Fanuc KAREL source: kb00143.KL

-- PROVISIONAL review KL for V1013-1; original PC SHA256 70a769824f0bb04e627808649afede2e4c1abad04249343c2b344672b59b27b0
-- Incomplete behavior may be omitted. Consult companion uncertainty JSON. Do not deploy.
PROGRAM KB00143
%NOLOCKGROUP
BEGIN
  -- UNRESOLVED_PC offsets 5-14; opcodes 3F,75
  -- UNRESOLVED_PC offsets 19-26; opcodes 9D,23
  -- UNRESOLVED_PC offsets 31-38; opcodes 9D,23
  -- UNRESOLVED_PC offsets 43-73; opcodes 27,22,2A,22,22,22,31
  -- UNRESOLVED_PC offsets 78-82; opcodes 7F
END KB00143
